// Mitsubishi GX Works2 project: FX1N   PLC: FX1N/FX1NC

// global labels: Global1
VAR_GLOBAL
  MainRun AT M0 : BOOL;
  MainRunI AT X001 : BOOL;
  MainStop AT M1 : BOOL;
  MainStopI AT X002 : BOOL;
  CoverRun AT M2 : BOOL;
  CoverRunI AT X006 : BOOL;
  SpinRun AT M3 : BOOL;
  SpinRunI AT X005 : BOOL;
  FlushRun AT M4 : BOOL;
  FlushRunI AT X015 : BOOL;
  CleanRun AT M5 : BOOL;
  CleanRunI AT X007 : BOOL;
  Mode AT D0 : INT;
  ModeManualI AT X003 : BOOL;
  ModeAutoI AT X004 : BOOL;
  MainState AT D1 : INT;
  MainStateNext AT M6 : BOOL;
  CoverState AT D2 : INT;
  CoverStateNext AT M7 : BOOL;
  SpinState AT D3 : INT;
  SpinStateNext AT M8 : BOOL;
  FlushState AT D4 : INT;
  FlushStateNext AT M9 : BOOL;
  CleanState AT D5 : INT;
  CleanStateNext AT M10 : BOOL;
  CoverPos AT D6 : INT;
  CoverUnlock AT M11 : BOOL;
  CoverUnlockO AT Y005 : BOOL;
  CoverUnlockN AT M12 : BOOL;
  CoverUnlockNTimer AT TC0 : BOOL;
  CoverUnlockNTimerDelay AT D128 : INT;
  CoverUnlockP AT M13 : BOOL;
  CoverUnlockPTimer AT TC1 : BOOL;
  CoverUnlockPTimerDelay AT D129 : INT;
  CoverNI AT X011 : BOOL;
  CoverNO AT Y006 : BOOL;
  CoverN AT M14 : BOOL;
  CoverNTimer AT TC2 : BOOL;
  CoverNTimerDelay AT D130 : INT;
  CoverPO AT Y007 : BOOL;
  CoverP AT M15 : BOOL;
  CoverPTimer AT TC3 : BOOL;
  CoverPTimerDelay AT D131 : INT;
  CoverFailTimer AT TC4 : BOOL;
  CoverFailTimerDelay AT D132 : INT;
  SpinPos AT D7 : INT;
  SpinUnlock AT M16 : BOOL;
  SpinUnlockN AT M17 : BOOL;
  SpinUnlockNTimer AT TC5 : BOOL;
  SpinUnlockNTimerDelay AT D133 : INT;
  SpinUnlockP AT M18 : BOOL;
  SpinUnlockPTimer AT TC6 : BOOL;
  SpinUnlockPTimerDelay AT D134 : INT;
  SpinBlock AT M19 : BOOL;
  SpinBlockN AT M20 : BOOL;
  SpinBlockNTimer AT TC7 : BOOL;
  SpinBlockNTimerDelay AT D135 : INT;
  SpinBlockP AT M21 : BOOL;
  SpinBlockPTimer AT TC8 : BOOL;
  SpinBlockPTimerDelay AT D136 : INT;
  SpinUnlockLO AT Y003 : BOOL;
  SpinUnlockRO AT Y004 : BOOL;
  SpinBlockO AT Y016 : BOOL;
  SpinP AT M22 : BOOL;
  SpinPI AT X010 : BOOL;
  SpinPO AT Y000 : BOOL;
  SpinBlockTimer AT TC9 : BOOL;
  SpinBlockTimerDelay AT D137 : INT;
  SpinFailTimer AT TC10 : BOOL;
  SpinFailTimerDelay AT D138 : INT;
  FlushEngage AT M23 : BOOL;
  FlushEngageO AT Y010 : BOOL;
  FlushEngageN AT M24 : BOOL;
  FlushEngageNTimer AT TC11 : BOOL;
  FlushEngageNTimerDelay AT D139 : INT;
  FlushEngageP AT M25 : BOOL;
  FlushEngagePTimer AT TC12 : BOOL;
  FlushEngagePTimerDelay AT D140 : INT;
  FlushTank AT M26 : BOOL;
  FlushTankO AT Y011 : BOOL;
  FlushTankN AT M27 : BOOL;
  FlushTankNTimer AT TC13 : BOOL;
  FlushTankNTimerDelay AT D141 : INT;
  FlushTankP AT M28 : BOOL;
  FlushTankPTimer AT TC14 : BOOL;
  FlushTankPTimerDelay AT D142 : INT;
  CleanPumpPos AT D8 : INT;
  CleanPumpO AT Y001 : BOOL;
  CleanPumpDirectionO AT Y012 : BOOL;
  CleanLowAI AT X012 : BOOL;
  CleanLowBI AT X013 : BOOL;
  CleanLowCI AT X014 : BOOL;
  CleanType AT D9 : INT;
  CleanTypeAO AT Y013 : BOOL;
  CleanTypeBO AT Y014 : BOOL;
  CleanTypeCO AT Y015 : BOOL;
  CleanSpreader AT M29 : BOOL;
  CleanSpreaderO AT Y002 : BOOL;
  CleanSprayTimer AT TC15 : ARRAY [0..4] OF BOOL;
  CleanSprayTimerDelay AT D143 : ARRAY [0..4] OF INT;
  CleanSoakTimer AT TC20 : ARRAY [0..4] OF BOOL;
  CleanSoakTimerDelay AT D148 : ARRAY [0..4] OF INT;
  ProblemExist AT M30 : BOOL;
  ProblemExistO AT Y017 : BOOL;
  ProblemIndex AT D10 : INT;
  Problem AT M600 : ARRAY [0..7] OF BOOL;
  TimeSetEnable AT M31 : BOOL;
  TimeSetTrigger AT M32 : BOOL;
  TimeBuffer AT D11 : ARRAY [0..6] OF INT;
  TimeYearIn AT D8018 : INT;
  TimeYear AT D18 : INT;
  TimeMonthIn AT D8017 : INT;
  TimeMonth AT D19 : INT;
  TimeDayIn AT D8016 : INT;
  TimeDay AT D20 : INT;
  TimeHourIn AT D8015 : INT;
  TimeHour AT D21 : INT;
  TimeMinIn AT D8014 : INT;
  TimeMin AT D22 : INT;
  TimeSecIn AT D8013 : INT;
  TimeSec AT D23 : INT;
  TimeOfWeekIn AT D8019 : INT;
  TimeOfWeek AT D24 : INT;
  ProcessDoorI AT X016 : BOOL;
  ProcessHumanI AT X017 : BOOL;
  ProcessHumanEnterFlushCount AT D25 : INT;
  ProcessHumanCount AT D153 : INT;
  ProcessHumanCountTimer AT TC25 : BOOL;
  ProcessHumanCountTimerDelay AT D154 : INT;
  ProcessFlushCount AT D155 : INT;
  ProcessCount AT D156 : INT;
  ProcessCountTarget AT D157 : INT;
  DecodeMode AT M33 : ARRAY [0..3] OF BOOL;
  DecodeCleanType AT M37 : ARRAY [0..3] OF BOOL;
END_VAR

// task Task_01 (event TRUE, interval 0, priority 31): POU_01

PROGRAM POU_01
VAR
  fTmp : BOOL;
  fRiseCover : BOOL;
  fFallCover : BOOL;
  fFirstRun : BOOL;
  fRiseFlush : BOOL;
  fRiseClean : BOOL;
  fRiseSpin : BOOL;
  fRiseRun : BOOL;
  fRiseStop : BOOL;
  fProblemFirst : BOOL;
  fHumanCountRise : BOOL;
  fHumanRise : BOOL;
  fHumanFall : BOOL;
  fHumanCountFlag : BOOL;
END_VAR
SET(M8002 AND CoverNTimerDelay <= 0, fTmp);
MOV(fTmp, 20, CoverUnlockNTimerDelay);
MOV(fTmp, 20, CoverUnlockPTimerDelay);
MOV(fTmp, 05, CoverNTimerDelay);
MOV(fTmp, 30, CoverPTimerDelay);
MOV(fTmp, 20, SpinUnlockNTimerDelay);
MOV(fTmp, 20, SpinUnlockPTimerDelay);
MOV(fTmp, 10, SpinBlockNTimerDelay);
MOV(fTmp, 10, SpinBlockPTimerDelay);
MOV(fTmp, 100, CleanSprayTimerDelay[0]);
MOV(fTmp, 101, CleanSprayTimerDelay[1]);
MOV(fTmp, 102, CleanSprayTimerDelay[2]);
MOV(fTmp, 103, CleanSprayTimerDelay[3]);
MOV(fTmp, 104, CleanSprayTimerDelay[4]);
MOV(fTmp, 10, CleanSoakTimerDelay[0]);
MOV(fTmp, 11, CleanSoakTimerDelay[1]);
MOV(fTmp, 12, CleanSoakTimerDelay[2]);
MOV(fTmp, 13, CleanSoakTimerDelay[3]);
MOV(fTmp, 14, CleanSoakTimerDelay[4]);
RST(fTmp, fTmp);
SET(M8002, MainStop);
SET(M8002, fFirstRun);
RST(M8002 AND ProcessCount < 0, ProcessCount);
RST(M8002 AND ProcessHumanCount < 0, ProcessHumanCount);
(*|||||||||||||||*)
(*|||||||||||||||*)
RST(M8002, TimeSetEnable);
RST(M8002, TimeSetTrigger);
TRD(M8000 AND NOT TimeSetEnable, TimeBuffer);
BMOV(M8000 AND NOT TimeSetEnable, TimeBuffer[0], 7, TimeYear);
SET(TimeSetEnable AND TimeSetTrigger, fTmp);
BMOV(fTmp, TimeYear, 7, TimeBuffer[0]);
TWR(fTmp, TimeBuffer);
RST(fTmp, TimeSetEnable);
RST(fTmp, TimeSetTrigger);
RST(fTmp, fTmp);
(*|||||||||||||||*)
(*|||||||||||||||*)
RST(ProblemExist, ProblemExist);
RST(M8000, ProblemIndex);
RST(fProblemFirst, fProblemFirst);
SET(Problem[0], ProblemExist);                                       SET(ProblemExist, fProblemFirst);
SET(Problem[1], ProblemExist); INC(NOT fProblemFirst, ProblemIndex); SET(ProblemExist, fProblemFirst);
SET(Problem[2], ProblemExist); INC(NOT fProblemFirst, ProblemIndex); SET(ProblemExist, fProblemFirst);
SET(Problem[3], ProblemExist); INC(NOT fProblemFirst, ProblemIndex); SET(ProblemExist, fProblemFirst);
SET(Problem[4], ProblemExist); INC(NOT fProblemFirst, ProblemIndex); SET(ProblemExist, fProblemFirst);
SET(Problem[5], ProblemExist); INC(NOT fProblemFirst, ProblemIndex); SET(ProblemExist, fProblemFirst);
SET(Problem[6], ProblemExist); INC(NOT fProblemFirst, ProblemIndex); SET(ProblemExist, fProblemFirst);
SET(Problem[7], ProblemExist); INC(NOT fProblemFirst, ProblemIndex); SET(ProblemExist, fProblemFirst);
(*|||||||||||||||*)
(*|||||||||||||||*)
SET(MainRun, fTmp);
RST(fTmp, MainRun);
MOV(fTmp, 1, MainState);
RST(fTmp, fTmp);
RST(MainRun, MainRun);
SET(MainStop, fTmp);
ZRST(fTmp, MainRun, CleanRun);
ZRST(fTmp, MainState, CleanState);
RST(fTmp, CoverUnlock);
RST(fTmp, CoverPos);
RST(fTmp, SpinUnlock);
RST(fTmp, SpinBlock);
RST(fTmp, SpinPos);
RST(fTmp, FlushEngage);
RST(fTmp, FlushTank);
RST(fTmp, CleanPumpPos);
RST(fTmp, CleanSpreader);
MOV(fTmp AND fFirstRun, 11, CoverState);
MOV(fTmp AND NOT fFirstRun AND CoverNI, 20, CoverState);
RST(fTmp AND fFirstRun, fFirstRun);
RST(fTmp, fTmp);
(*||||||||||||||||*)
(*|||||DECODE|||||*)
(*||||||||||||||||*)
INC(MainStateNext, MainState);
INC(CoverStateNext, CoverState);
INC(SpinStateNext, SpinState);
INC(FlushStateNext, FlushState);
INC(CleanStateNext, CleanState);
ZRST(M8000, MainStateNext, CleanStateNext);
DECO(M8000, MainState,  6, M100);
DECO(M8000, CoverState, 6, M200);
DECO(M8000, SpinState,  6, M300);
DECO(M8000, FlushState, 6, M400);
DECO(M8000, CleanState, 6, M500);
(**)
DECO(M8000, Mode, 2, DecodeMode[0]);
DECO(M8000, CleanType, 2, DecodeCleanType[0]);
(*||||||||||||||*)
(*|||||MAIN|||||*)
(*||||||||||||||*)
(*uncover*)
SET(M101, fTmp);
MOV(fTmp, 11, CoverState);
SET(fTmp, MainStateNext);
RST(fTmp, fTmp);
(*uncover done -> spin*)
SET(M102 AND M220, fTmp);
MOV(fTmp, 1, SpinState);
SET(fTmp, MainStateNext);
RST(fTmp, fTmp);
(*spin done -> cover, flush*)
SET(M103 AND M300, fTmp);
MOV(fTmp, 1, CoverState);
MOV(fTmp, 1, FlushState);
SET(fTmp, MainStateNext);
RST(fTmp, fTmp);
(*cover done -> clean*)
SET(M104 AND M210, fTmp);
MOV(fTmp, 1, CleanState);
SET(fTmp, MainStateNext);
RST(fTmp, fTmp);
(*flush, clean done -> uncover*)
SET(M105 AND M400 AND M500, fTmp);
MOV(fTmp, 11, CoverState);
SET(fTmp, MainStateNext);
RST(fTmp, fTmp);
(*uncover done -> end*)
SET(M106 AND M220, fTmp);
RST(fTmp, ProcessCount);
RST(fTmp, MainState);
RST(fTmp, fTmp);
(*|||||||||||||||*)
(*|||||COVER|||||*)
(*|||||||||||||||*)
(*-DOWN-*)
(*unlock*)
MOV(M201 AND NOT CoverNI, 6, CoverState);
SET(M201 AND CoverNI, fTmp);
MOV(fTmp, -1, CoverPos);
SET(fTmp, CoverUnlock);
SET(fTmp, CoverStateNext);
RST(fTmp, fTmp);
(*unlock done -> move down*)
SET(M202 AND CoverUnlockN, fTmp);
MOV(fTmp, 1, CoverPos);
SET(fTmp, CoverStateNext);
RST(fTmp, fTmp);
(*move down done -> end*)
SET(M203 AND CoverP, fTmp);
RST(fTmp, CoverUnlock);
RST(fTmp, CoverPos);
MOV(fTmp, 10, CoverState);
RST(fTmp, fTmp);
(*early exit*)
SET(M206, fTmp);
MOV(fTmp, 1, CoverPos);
MOV(fTmp, 3, CoverState);
RST(fTmp, fTmp);
(*-UP-*)
(*unlock*)
MOV(M211 AND CoverNI, 15, CoverState);
SET(M211 AND NOT CoverNI, fTmp);
SET(fTmp, CoverUnlock);
SET(fTmp, CoverStateNext);
RST(fTmp, fTmp);
(*unlock done -> move up*)
SET(M212 AND CoverUnlockN, fTmp);
MOV(fTmp, -1, CoverPos);
SET(fTmp, CoverStateNext);
RST(fTmp, fTmp);
(*move up done -> lock*)
OUT_T(M213, CoverFailTimer, CoverFailTimerDelay);
MOV(M213 AND CoverFailTimer, 21, CoverState);
SET(M213 AND CoverN, fTmp);
RST(fTmp, CoverUnlock);
SET(fTmp, CoverStateNext);
RST(fTmp, fTmp);
(*lock done -> end*)
SET(M214 AND CoverUnlockP, fTmp);
RST(fTmp, CoverPos);
MOV(fTmp, 20, CoverState);
RST(fTmp, fTmp);
(*early exit*)
SET(M215, fTmp);
MOV(fTmp, -1, CoverPos);
MOV(fTmp, 13, CoverState);
RST(fTmp, fTmp);
(*fail -> wait retry*)
SET(M221, fTmp);
RST(fTmp, CoverUnlock);
RST(fTmp, CoverPos);
SET(fTmp, ProblemExist);
SET(fTmp, Problem[0]);
SET(fTmp, CoverStateNext);
RST(fTmp, fTmp);
(*wait retry -> retry*)
SET(M222 AND NOT Problem[0], fTmp);
MOV(fTmp, 11, CoverState);
RST(fTmp, fTmp);
(*||||||||||||||*)
(*|||||SPIN|||||*)
(*||||||||||||||*)
(*unlock, unblock*)
SET(M301, fTmp);
SET(fTmp, SpinUnlock);
RST(fTmp, SpinBlock);
SET(fTmp, SpinStateNext);
RST(fTmp, fTmp);
(*unlock, unblock done -> spin*)
SET(M302 AND SpinUnlockN AND SpinBlockN, fTmp);
MOV(fTmp, 1, SpinPos);
RST(fTmp, SpinP);
SET(fTmp, SpinStateNext);
RST(fTmp, fTmp);
(*wait -> block*)
OUT_T(M303 AND NOT SpinPI, SpinBlockTimer, SpinBlockTimerDelay);
SET(M303 AND SpinBlockTimer, fTmp);
SET(fTmp, SpinBlock);
SET(fTmp, SpinStateNext);
RST(fTmp, fTmp);
(*sensor rise -> stop*)
OUT_T(M304, SpinFailTimer, SpinFailTimerDelay);
MOV(M304 AND SpinFailTimer, 11, SpinState);
SET(M304 AND SpinP, fTmp);
RST(fTmp, SpinPos);
SET(fTmp, SpinStateNext);
RST(fTmp, fTmp);
(*stop done -> lock*)
SET(M305, fTmp);
RST(fTmp, SpinUnlock);
SET(fTmp, SpinStateNext);
RST(fTmp, fTmp);
(*lock done -> end*)
SET(M306 AND SpinUnlockP, fTmp);
RST(fTmp, SpinBlock);
RST(fTmp, SpinState);
RST(fTmp, fTmp);
(*fail -> wait retry*)
SET(M311, fTmp);
RST(fTmp, SpinPos);
SET(fTmp, ProblemExist);
SET(fTmp, Problem[1]);
SET(fTmp, SpinStateNext);
RST(fTmp, fTmp);
(*wait retry -> retry*)
SET(M312 AND NOT Problem[1], fTmp);
MOV(fTmp, 1, SpinState);
RST(fTmp, fTmp);
(*|||||||||||||||*)
(*|||||FLUSH|||||*)
(*|||||||||||||||*)
(*engage*)
SET(M401, fTmp);
SET(fTmp, FlushEngage);
RST(fTmp, FlushTank);
SET(fTmp, FlushStateNext);
RST(fTmp, fTmp);
(*flush*)
SET(M402 AND FlushEngageP AND FlushTankN, fTmp);
SET(fTmp, FlushTank);
SET(fTmp, FlushStateNext);
RST(fTmp, fTmp);
(*unflush*)
SET(M403 AND FlushTankP, fTmp);
RST(fTmp, FlushTank);
SET(fTmp, FlushStateNext);
RST(fTmp, fTmp);
(*unengage*)
SET(M404 AND FlushTankN, fTmp);
RST(fTmp, FlushEngage);
SET(fTmp, FlushStateNext);
RST(fTmp, fTmp);
(*done*)
SET(M405 AND FlushEngageN, fTmp);
INC(fTmp, ProcessFlushCount);
RST(fTmp, FlushState);
RST(fTmp, fTmp);
(*|||||||||||||||*)
(*|||||CLEAN|||||*)
(*|||||||||||||||*)
(*start*)
SET(M501, fTmp);
SET(fTmp, CleanSpreader);
SET(fTmp, CleanStateNext);
RST(fTmp, fTmp);
(*0*)
(*spray*)
SET(M502, fTmp);
MOV(fTmp, 1, CleanPumpPos);
MOV(fTmp, 0, CleanType);
SET(fTmp, CleanStateNext);
RST(fTmp, fTmp);
(*spray done -> soak*)
OUT_T(M503, CleanSprayTimer[0], CleanSprayTimerDelay[0]);
SET(M503 AND CleanSprayTimer[0], fTmp);
RST(fTmp, CleanPumpPos);
SET(fTmp, CleanStateNext);
RST(fTmp, fTmp);
(*soak done*)
OUT_T(M504, CleanSoakTimer[0], CleanSoakTimerDelay[0]);
SET(M504 AND CleanSoakTimer[0], fTmp);
SET(fTmp, CleanStateNext);
RST(fTmp, fTmp);
(*1*)
(*spray*)
SET(M505, fTmp);
MOV(fTmp, 1, CleanPumpPos);
MOV(fTmp, 1, CleanType);
SET(fTmp, CleanStateNext);
RST(fTmp, fTmp);
(*spray done -> soak*)
OUT_T(M506, CleanSprayTimer[1], CleanSprayTimerDelay[1]);
SET(M506 AND CleanSprayTimer[1], fTmp);
RST(fTmp, CleanPumpPos);
SET(fTmp, CleanStateNext);
RST(fTmp, fTmp);
(*soak done*)
OUT_T(M507, CleanSoakTimer[1], CleanSoakTimerDelay[1]);
SET(M507 AND CleanSoakTimer[1], fTmp);
SET(fTmp, CleanStateNext);
RST(fTmp, fTmp);
(*2*)
(*spray*)
SET(M508, fTmp);
MOV(fTmp, 1, CleanPumpPos);
MOV(fTmp, 2, CleanType);
SET(fTmp, CleanStateNext);
RST(fTmp, fTmp);
(*spray done -> soak*)
OUT_T(M509, CleanSprayTimer[2], CleanSprayTimerDelay[2]);
SET(M509 AND CleanSprayTimer[2], fTmp);
RST(fTmp, CleanPumpPos);
SET(fTmp, CleanStateNext);
RST(fTmp, fTmp);
(*soak done*)
OUT_T(M510, CleanSoakTimer[2], CleanSoakTimerDelay[2]);
SET(M510 AND CleanSoakTimer[2], fTmp);
SET(fTmp, CleanStateNext);
RST(fTmp, fTmp);
(*3*)
(*spray*)
SET(M511, fTmp);
MOV(fTmp, 1, CleanPumpPos);
MOV(fTmp, 0, CleanType);
SET(fTmp, CleanStateNext);
RST(fTmp, fTmp);
(*spray done -> soak*)
OUT_T(M512, CleanSprayTimer[3], CleanSprayTimerDelay[3]);
SET(M512 AND CleanSprayTimer[3], fTmp);
RST(fTmp, CleanPumpPos);
SET(fTmp, CleanStateNext);
RST(fTmp, fTmp);
(*soak done*)
OUT_T(M513, CleanSoakTimer[3], CleanSoakTimerDelay[3]);
SET(M513 AND CleanSoakTimer[3], fTmp);
SET(fTmp, CleanStateNext);
RST(fTmp, fTmp);
(*4*)
(*spray*)
SET(M514, fTmp);
MOV(fTmp, 2, CleanPumpPos);
MOV(fTmp, 0, CleanType);
SET(fTmp, CleanStateNext);
RST(fTmp, fTmp);
(*spray done -> soak*)
OUT_T(M515, CleanSprayTimer[4], CleanSprayTimerDelay[4]);
SET(M515 AND CleanSprayTimer[4], fTmp);
RST(fTmp, CleanPumpPos);
SET(fTmp, CleanStateNext);
RST(fTmp, fTmp);
(*soak done*)
OUT_T(M516, CleanSoakTimer[4], CleanSoakTimerDelay[4]);
SET(M516 AND CleanSoakTimer[4], fTmp);
SET(fTmp, CleanStateNext);
RST(fTmp, fTmp);
(*done*)
SET(M517, fTmp);
RST(fTmp, CleanPumpPos);
RST(fTmp, CleanType);
RST(fTmp, CleanSpreader);
RST(fTmp, CleanState);
RST(fTmp, fTmp);
(*|||||||||||||||*)
(*|||||INPUT|||||*)
(*|||||||||||||||*)
PLS(MainRunI, fRiseRun);   SET(fRiseRun, MainRun);
PLF(MainStopI, fRiseStop); SET(fRiseStop, MainStop);
RST(M8000, Mode); MOV(ModeManualI, 1, Mode); MOV(ModeAutoI, 2, Mode);
PLS(CoverRunI, fRiseCover); SET(fRiseCover, CoverRun); MOV(DecodeMode[1] AND CoverRun AND M100 AND (M200 OR M220), 01, CoverState);                  RST(CoverRun, CoverRun);
PLF(CoverRunI, fFallCover); SET(fFallCover, CoverRun); MOV(DecodeMode[1] AND CoverRun AND M100 AND (M200 OR M210), 11, CoverState);                  RST(CoverRun, CoverRun);
PLS(SpinRunI, fRiseSpin);   SET(fRiseSpin, SpinRun);   MOV(DecodeMode[1] AND SpinRun AND M100 AND M220 AND M300 AND M400, 01, SpinState);            RST(SpinRun, SpinRun);
PLS(FlushRunI, fRiseFlush); SET(fRiseFlush, FlushRun); MOV(FlushRun AND M100 AND M300 AND M400, 01, FlushState);                                     RST(FlushRun, FlushRun);
PLS(CleanRunI, fRiseClean); SET(fRiseClean, CleanRun); MOV(DecodeMode[1] AND CleanRun AND M100 AND M210 AND M300 AND M400 AND M500, 01, CleanState); RST(CleanRun, CleanRun);
PLS(SpinPI, SpinP);         SET(SpinP, SpinP);
SET(CleanLowAI, Problem[2]);
SET(CleanLowBI, Problem[3]);
SET(CleanLowCI, Problem[4]);
(**)
RST(CoverUnlockN, CoverUnlockN); RST(CoverUnlockP, CoverUnlockP);
RST(CoverN, CoverN);             RST(CoverP, CoverP);
RST(SpinUnlockN, SpinUnlockN);   RST(SpinUnlockP, SpinUnlockP);
RST(SpinBlockN, SpinBlockN);     RST(SpinBlockP, SpinBlockP);
RST(FlushEngageN, FlushEngageN); RST(FlushEngageP, FlushEngageP);
RST(FlushTankN, FlushTankN);     RST(FlushTankP, FlushTankP);
(**)
OUT_T(CoverUnlock,              CoverUnlockNTimer, CoverUnlockNTimerDelay); SET(CoverUnlockNTimer, CoverUnlockN); RST(CoverUnlockNTimer, CoverUnlockP);
OUT_T(NOT CoverUnlock,          CoverUnlockPTimer, CoverUnlockPTimerDelay); SET(CoverUnlockPTimer, CoverUnlockP); RST(CoverUnlockPTimer, CoverUnlockN);
OUT_T(CoverPos < 0 AND CoverNI, CoverNTimer, CoverNTimerDelay);             SET(CoverNTimer, CoverN);             RST(CoverNTimer, CoverP);
OUT_T(CoverPos > 0,             CoverPTimer, CoverPTimerDelay);             SET(CoverPTimer, CoverP);             RST(CoverPTimer, CoverN);
OUT_T(SpinUnlock,               SpinUnlockNTimer, SpinUnlockNTimerDelay);   SET(SpinUnlockNTimer, SpinUnlockN);   RST(SpinUnlockNTimer, SpinUnlockP);
OUT_T(NOT SpinUnlock,           SpinUnlockPTimer, SpinUnlockPTimerDelay);   SET(SpinUnlockPTimer, SpinUnlockP);   RST(SpinUnlockPTimer, SpinUnlockN);
OUT_T(NOT SpinBlock,            SpinBlockNTimer, SpinBlockNTimerDelay);     SET(SpinBlockNTimer, SpinBlockN);     RST(SpinBlockNTimer, SpinBlockP);
OUT_T(SpinBlock,                SpinBlockPTimer, SpinBlockPTimerDelay);     SET(SpinBlockPTimer, SpinBlockP);     RST(SpinBlockPTimer, SpinBlockN);
OUT_T(NOT FlushEngage,          FlushEngageNTimer, FlushEngageNTimerDelay); SET(FlushEngageNTimer, FlushEngageN); RST(FlushEngageNTimer, FlushEngageP);
OUT_T(FlushEngage,              FlushEngagePTimer, FlushEngagePTimerDelay); SET(FlushEngagePTimer, FlushEngageP); RST(FlushEngagePTimer, FlushEngageN);
OUT_T(NOT FlushTank,            FlushTankNTimer, FlushTankNTimerDelay);     SET(FlushTankNTimer, FlushTankN);     RST(FlushTankNTimer, FlushTankP);
OUT_T(FlushTank,                FlushTankPTimer, FlushTankPTimerDelay);     SET(FlushTankPTimer, FlushTankP);     RST(FlushTankPTimer, FlushTankN);
(**)
PLS(ProcessHumanI, fHumanRise); SET(fHumanRise, fTmp);
MOV(fTmp, ProcessFlushCount, ProcessHumanEnterFlushCount);
RST(fTmp, fHumanCountFlag);
RST(fTmp, fTmp);
OUT_T(ProcessHumanI, ProcessHumanCountTimer, ProcessHumanCountTimerDelay);
PLS(ProcessHumanCountTimer, fHumanCountRise); SET(fHumanCountRise, fHumanCountFlag);
PLF(ProcessHumanI, fHumanFall); SET(fHumanFall, fTmp);
RST(NOT fHumanCountFlag, fTmp);
INC(fTmp, ProcessHumanCount);
SET(fTmp AND ProcessFlushCount = ProcessHumanEnterFlushCount, FlushRun);
RST(fTmp, ProcessFlushCount);
INC(fTmp, ProcessCount);
RST(fTmp, fTmp);
SET(ProcessDoorI AND ProcessCount >= ProcessCountTarget AND NOT (ProcessHumanI OR FlushRun), MainRun);
RST(MainRun AND NOT (M100 AND DecodeMode[2]), MainRun);
(*||||||||||||||||*)
(*|||||OUTPUT|||||*)
(*||||||||||||||||*)
OUT(CoverUnlock, CoverUnlockO);
OUT(CoverPos < 0, CoverNO);
OUT(CoverPos > 0, CoverPO);
OUT(SpinUnlock, SpinUnlockLO);
OUT(SpinUnlock, SpinUnlockRO);
OUT(SpinBlock, SpinBlockO);
OUT(SpinPos > 0, SpinPO);
OUT(FlushEngage, FlushEngageO);
OUT(FlushTank, FlushTankO);
(**)
OUT(CleanPumpPos > 0, CleanPumpO);
RST(CleanLowAI AND DecodeCleanType[0], CleanPumpO);
RST(CleanLowBI AND DecodeCleanType[1], CleanPumpO);
RST(CleanLowCI AND DecodeCleanType[2], CleanPumpO);
(**)
OUT(CleanPumpO AND CleanPumpPos = 2, CleanPumpDirectionO);
OUT(CleanPumpO AND DecodeCleanType[0], CleanTypeAO);
OUT(CleanPumpO AND DecodeCleanType[1], CleanTypeBO);
OUT(CleanPumpO AND DecodeCleanType[2], CleanTypeCO);
OUT(CleanSpreader, CleanSpreaderO);
(*|||||||||||||||*)
END_PROGRAM
